Staubli VAL3: multi.pgx

program multi()
begin
do
//getting the joint variables
jAxis=herej()
nAxis[0]=jAxis.j1
nAxis[1]=jAxis.j2
nAxis[2]=jAxis.j3
nAxis[3]=jAxis.j4
nAxis[4]=jAxis.j5
nAxis[5]=jAxis.j6
//saving all data to one binary package
toBinary(nAxis, 6, "8.0b", nByteOut)
//sending to defined address.
sioSet(sCal, nByteOut)
delay(0)
until (bEnd==true)
end
